DATA_BLOCK "起动过程_DB"
{ S7_Optimized_Access := 'TRUE' }
VERSION : 0.1
NON_RETAIN
"起动过程"

BEGIN

END_DATA_BLOCK

